% RSLogix 500 project MotorStarter.RSS, saved by version 8.30.00.16 %
PROJECT "UNTITLED"    % processor: Bul.1763 MicroLogix 1100 Series B %

PROGRAM FILES
  LAD 2   3 rungs

DATA FILES
  O0 OUTPUT  4 elements
  I1 INPUT  6 elements
  S2 STATUS  66 elements
  B3 BINARY  10 elements
  T4 TIMER  1 elements
  C5 COUNTER  1 elements
  R6 CONTROL  1 elements
  N7 INTEGER  1 elements
  F8 FLOAT  1 elements

LADDER 2
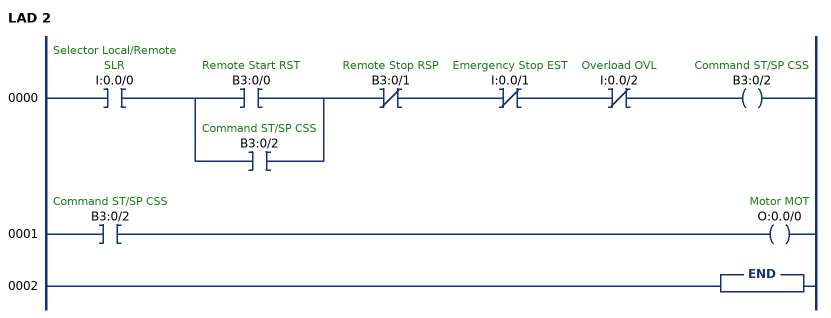
% Rung: 0 %
SOR XIC I:0.0/0 BST XIC B3:0/0 NXB XIC B3:0/2 BND XIO B3:0/1 XIO I:0.0/1 XIO I:0.0/2 OTE B3:0/2 EOR
%   I:0.0/0  SLR  "Selector Local/Remote" %
%   B3:0/0  RST  "Remote Start" %
%   B3:0/2  CSS  "Command ST/SP" %
%   B3:0/1  RSP  "Remote Stop" %
%   I:0.0/1  EST  "Emergency Stop" %
%   I:0.0/2  OVL  "Overload" %
% Rung: 1 %
SOR XIC B3:0/2 OTE O:0.0/0 EOR
%   B3:0/2  CSS  "Command ST/SP" %
%   O:0.0/0  MOT  "Motor" %
% Rung: 2 %
SOR END EOR

DATA TABLE (non-zero values as saved)
DATA B3
% B3:0 % 0X0005 0X0000 0X0000 0X0000 0X0000 0X0000 0X0000 0X0000 0X0000 0X0000
